DATA_BLOCK "Zne04_DB"
{ S7_Optimized_Access := 'TRUE' }
VERSION : 0.1
NON_RETAIN
"Zne04"

BEGIN

END_DATA_BLOCK

